LIN {X 0,Y 60.653,Z 1002.09,A -85,B 0,C 180,E1 2720.013,E2 2720.013} C_VEL
LIN {X 0,Y 76.749,Z 998.307,A -85,B 0,C 180,E1 2712.299,E2 2712.299} C_VEL
LIN {X 0,Y 92.827,Z 993.043,A -85,B 0,C 180,E1 2707.719,E2 2707.719} C_VEL
LIN {X 0,Y 109.349,Z 985.916,A -85,B 0,C 180,E1 2704.684,E2 2704.684} C_VEL
LIN {X 0,Y 120.443,Z 980.063,A -85,B 0,C 180,E1 2703.187,E2 2703.187} C_VEL
LIN {X 0,Y 109.037,Z 985.343,A -85,B 0,C 180,E1 2701.127,E2 2701.127} C_VEL
LIN {X 0,Y 102.027,Z 988.229,A -85,B 0,C 180,E1 2700.205,E2 2700.205} C_VEL
LIN {X 0,Y 85.588,Z 993.654,A -85,B 0,C 180,E1 2699.608,E2 2699.608} C_VEL
LIN {X 0,Y 77.632,Z 995.551,A -85,B 0,C 180,E1 2698.509,E2 2698.509} C_VEL
LIN {X 0,Y 75.592,Z 995.92,A -85,B 0,C 180,E1 2697.928,E2 2697.928} C_VEL
LIN {X 0,Y 59.701,Z 997.838,A -85,B 0,C 180,E1 2691.151,E2 2691.151} C_VEL
LIN {X 0,Y 45.629,Z 997.877,A -85,B 0,C 180,E1 2680.427,E2 2680.427} C_VEL
LIN {X 0,Y 33.755,Z 996.072,A -85,B 0,C 180,E1 2660.363,E2 2660.363} C_VEL
LIN {X 0,Y 28.785,Z 992.656,A -85,B 0,C 180,E1 2630.292,E2 2630.292} C_VEL
LIN {X 0,Y 32.409,Z 987.446,A -85,B 0,C 180,E1 2599.329,E2 2599.329} C_VEL
LIN {X 0,Y 42.338,Z 980.363,A -85,B 0,C 180,E1 2578.694,E2 2578.694} C_VEL
LIN {X 0,Y 54.402,Z 971.765,A -85,B 0,C 180,E1 2567.152,E2 2567.152} C_VEL
LIN {X 0,Y 66.783,Z 961.6,A -85,B 0,C 180,E1 2560.218,E2 2560.218} C_VEL
LIN {X 0,Y 78.97,Z 949.788,A -85,B 0,C 180,E1 2555.623,E2 2555.623} C_VEL
LIN {X 0,Y 89.724,Z 937.203,A -85,B 0,C 180,E1 2552.576,E2 2552.576} C_VEL
LIN {X 0,Y 99.614,Z 923.075,A -85,B 0,C 180,E1 2550.318,E2 2550.318} C_VEL
LIN {X 0,Y 108.255,Z 907.797,A -85,B 0,C 180,E1 2548.663,E2 2548.663} C_VEL
LIN {X 0,Y 114.969,Z 892.51,A -85,B 0,C 180,E1 2547.49,E2 2547.49} C_VEL
LIN {X 0,Y 120.607,Z 875.116,A -85,B 0,C 180,E1 2546.545,E2 2546.545} C_VEL
LIN {X 0,Y 124.343,Z 857.735,A -85,B 0,C 180,E1 2545.892,E2 2545.892} C_VEL
LIN {X 0,Y 132.685,Z 790.079,A -85,B 0,C 180,E1 2544.548,E2 2544.548} C_VEL
LIN {X 0,Y 132.195,Z 786.817,A -85,B 0,C 180,E1 2541.513,E2 2541.513} C_VEL
LIN {X 0,Y 131.977,Z 784.886,A -85,B 0,C 180,E1 2539.013,E2 2539.013} C_VEL
LIN {X 0,Y 131.942,Z 783.505,A -85,B 0,C 180,E1 2534.932,E2 2534.932} C_VEL
LIN {X 0,Y 132.207,Z 783.997,A -85,B 0,C 180,E1 2531.12,E2 2531.12} C_VEL
LIN {X 0,Y 132.675,Z 785.81,A -85,B 0,C 180,E1 2528.015,E2 2528.015} C_VEL
LIN {X 0,Y 133.455,Z 788.917,A -85,B 0,C 180,E1 2524.728,E2 2524.728} C_VEL
LIN {X 0,Y 133.681,Z 790.106,A -85,B 0,C 180,E1 2523.881,E2 2523.881} C_VEL
LIN {X 0,Y 124.607,Z 863.761,A -85,B 0,C 180,E1 2522.537,E2 2522.537} C_VEL
LIN {X 0,Y 120.434,Z 881.969,A -85,B 0,C 180,E1 2522.002,E2 2522.002} C_VEL
LIN {X 0,Y 115.02,Z 897.971,A -85,B 0,C 180,E1 2521.383,E2 2521.383} C_VEL
LIN {X 0,Y 107.621,Z 914.175,A -85,B 0,C 180,E1 2520.533,E2 2520.533} C_VEL
LIN {X 0,Y 98.541,Z 929.75,A -85,B 0,C 180,E1 2519.263,E2 2519.263} C_VEL
LIN {X 0,Y 88.081,Z 944.264,A -85,B 0,C 180,E1 2517.398,E2 2517.398} C_VEL
LIN {X 0,Y 76.332,Z 957.549,A -85,B 0,C 180,E1 2514.586,E2 2514.586} C_VEL
LIN {X 0,Y 63.894,Z 969.277,A -85,B 0,C 180,E1 2510.371,E2 2510.371} C_VEL
LIN {X 0,Y 51.107,Z 979.561,A -85,B 0,C 180,E1 2503.47,E2 2503.47} C_VEL
LIN {X 0,Y 38.783,Z 988.262,A -85,B 0,C 180,E1 2491.235,E2 2491.235} C_VEL
LIN {X 0,Y 29.178,Z 995.42,A -85,B 0,C 180,E1 2467.992,E2 2467.992} C_VEL
LIN {X 0,Y 27.175,Z 1000.596,A -85,B 0,C 180,E1 2434.224,E2 2434.224} C_VEL
LIN {X 0,Y 27.841,Z 1001.338,A -85,B 0,C 180,E1 2427.946,E2 2427.946} C_VEL
LIN {X 0,Y 30.091,Z 1003.083,A -85,B 0,C 180,E1 2388.356,E2 2388.356} C_VEL
LIN {X 0,Y 42.638,Z 1002.936,A -85,B 0,C 180,E1 2363.864,E2 2363.864} C_VEL
LIN {X 0,Y 59.278,Z 1000.831,A -85,B 0,C 180,E1 2351.965,E2 2351.965} C_VEL
LIN {X 0,Y 77.369,Z 996.828,A -85,B 0,C 180,E1 2345.69,E2 2345.69} C_VEL
LIN {X 0,Y 92.858,Z 991.915,A -85,B 0,C 180,E1 2342.506,E2 2342.506} C_VEL
LIN {X 0,Y 77.018,Z 995.662,A -85,B 0,C 180,E1 2338.389,E2 2338.389} C_VEL
LIN {X 0,Y 75.592,Z 995.92,A -85,B 0,C 180,E1 2337.928,E2 2337.928} C_VEL
LIN {X 0,Y 68.255,Z 997.161,A -85,B 0,C 180,E1 2336.138,E2 2336.138} C_VEL
LIN {X 0,Y 51.751,Z 999.008,A -85,B 0,C 180,E1 2333.791,E2 2333.791} C_VEL
LIN {X 0,Y 43.257,Z 999.163,A -85,B 0,C 180,E1 2330.629,E2 2330.629} C_VEL
LIN {X 0,Y 41.305,Z 999.049,A -85,B 0,C 180,E1 2329.203,E2 2329.203} C_VEL
LIN {X 0,Y 27.352,Z 997.144,A -85,B 0,C 180,E1 2309.214,E2 2309.214} C_VEL
LIN {X 0,Y 20.883,Z 993.753,A -85,B 0,C 180,E1 2272.517,E2 2272.517} C_VEL
LIN {X 0,Y 25.444,Z 988.485,A -85,B 0,C 180,E1 2231.673,E2 2231.673} C_VEL
LIN {X 0,Y 37.244,Z 981.364,A -85,B 0,C 180,E1 2209.882,E2 2209.882} C_VEL
LIN {X 0,Y 49.819,Z 973.257,A -85,B 0,C 180,E1 2199.962,E2 2199.962} C_VEL
LIN {X 0,Y 62.789,Z 963.343,A -85,B 0,C 180,E1 2194.097,E2 2194.097} C_VEL
LIN {X 0,Y 75.306,Z 951.859,A -85,B 0,C 180,E1 2190.338,E2 2190.338} C_VEL
LIN {X 0,Y 86.989,Z 938.866,A -85,B 0,C 180,E1 2187.739,E2 2187.739} C_VEL
LIN {X 0,Y 97.26,Z 924.717,A -85,B 0,C 180,E1 2185.901,E2 2185.901} C_VEL
LIN {X 0,Y 106.1,Z 909.608,A -85,B 0,C 180,E1 2184.575,E2 2184.575} C_VEL
LIN {X 0,Y 112.962,Z 894.711,A -85,B 0,C 180,E1 2183.634,E2 2183.634} C_VEL
LIN {X 0,Y 118.75,Z 877.722,A -85,B 0,C 180,E1 2182.859,E2 2182.859} C_VEL
LIN {X 0,Y 122.816,Z 860.067,A -85,B 0,C 180,E1 2182.285,E2 2182.285} C_VEL
LIN {X 0,Y 130.037,Z 803.511,A -85,B 0,C 180,E1 2181.336,E2 2181.336} C_VEL
LIN {X 0,Y 131.077,Z 794.946,A -85,B 0,C 180,E1 2181.139,E2 2181.139} C_VEL
LIN {X 0,Y 130.91,Z 792.632,A -85,B 0,C 180,E1 2178.25,E2 2178.25} C_VEL
LIN {X 0,Y 130.947,Z 791.448,A -85,B 0,C 180,E1 2174.595,E2 2174.595} C_VEL
LIN {X 0,Y 131.157,Z 791.938,A -85,B 0,C 180,E1 2171.433,E2 2171.433} C_VEL
LIN {X 0,Y 131.529,Z 793.772,A -85,B 0,C 180,E1 2168.526,E2 2168.526} C_VEL
LIN {X 0,Y 131.748,Z 795.084,A -85,B 0,C 180,E1 2167.209,E2 2167.209} C_VEL
LIN {X 0,Y 123.138,Z 863.302,A -85,B 0,C 180,E1 2166.178,E2 2166.178} C_VEL
LIN {X 0,Y 118.848,Z 881.619,A -85,B 0,C 180,E1 2165.757,E2 2165.757} C_VEL
LIN {X 0,Y 112.966,Z 898.485,A -85,B 0,C 180,E1 2165.279,E2 2165.279} C_VEL
LIN {X 0,Y 105.338,Z 914.598,A -85,B 0,C 180,E1 2164.672,E2 2164.672} C_VEL
LIN {X 0,Y 96.197,Z 929.815,A -85,B 0,C 180,E1 2163.771,E2 2163.771} C_VEL
LIN {X 0,Y 85.566,Z 944.072,A -85,B 0,C 180,E1 2162.411,E2 2162.411} C_VEL
LIN {X 0,Y 73.493,Z 957.227,A -85,B 0,C 180,E1 2160.305,E2 2160.305} C_VEL
LIN {X 0,Y 60.081,Z 969.265,A -85,B 0,C 180,E1 2156.913,E2 2156.913} C_VEL
LIN {X 0,Y 46.541,Z 979.31,A -85,B 0,C 180,E1 2151.224,E2 2151.224} C_VEL
LIN {X 0,Y 32.97,Z 987.831,A -85,B 0,C 180,E1 2140.082,E2 2140.082} C_VEL
LIN {X 0,Y 21.61,Z 994.812,A -85,B 0,C 180,E1 2113.957,E2 2113.957} C_VEL
LIN {X 0,Y 19.732,Z 999.841,A -85,B 0,C 180,E1 2066.737,E2 2066.737} C_VEL
LIN {X 0,Y 23.96,Z 1001.639,A -85,B 0,C 180,E1 2017.55,E2 2017.55} C_VEL
LIN {X 0,Y 39.12,Z 1001.702,A -85,B 0,C 180,E1 1993.786,E2 1993.786} C_VEL
LIN {X 0,Y 57.155,Z 999.903,A -85,B 0,C 180,E1 1984.344,E2 1984.344} C_VEL
LIN {X 0,Y 66.019,Z 998.339,A -85,B 0,C 180,E1 1981.724,E2 1981.724} C_VEL
LIN {X 0,Y 50.166,Z 999.311,A -85,B 0,C 180,E1 1975.222,E2 1975.222} C_VEL
LIN {X 0,Y 41.305,Z 999.049,A -85,B 0,C 180,E1 1969.203,E2 1969.203} C_VEL
LIN {X 0,Y 34.357,Z 998.611,A -85,B 0,C 180,E1 1963.944,E2 1963.944} C_VEL
LIN {X 0,Y 20.106,Z 997.162,A -85,B 0,C 180,E1 1949.983,E2 1949.983} C_VEL
LIN {X 0,Y 13.717,Z 995.406,A -85,B 0,C 180,E1 1926.437,E2 1926.437} C_VEL
LIN {X 0,Y 12.976,Z 994.699,A -85,B 0,C 180,E1 1915.311,E2 1915.311} C_VEL
LIN {X 0,Y 19.259,Z 989.522,A -85,B 0,C 180,E1 1858.718,E2 1858.718} C_VEL
LIN {X 0,Y 33.288,Z 982.367,A -85,B 0,C 180,E1 1838.646,E2 1838.646} C_VEL
LIN {X 0,Y 46.778,Z 974.342,A -85,B 0,C 180,E1 1831.237,E2 1831.237} C_VEL
LIN {X 0,Y 60.595,Z 964.276,A -85,B 0,C 180,E1 1826.991,E2 1826.991} C_VEL
LIN {X 0,Y 73.542,Z 952.771,A -85,B 0,C 180,E1 1824.363,E2 1824.363} C_VEL
LIN {X 0,Y 85.525,Z 939.759,A -85,B 0,C 180,E1 1822.541,E2 1822.541} C_VEL
LIN {X 0,Y 96.011,Z 925.604,A -85,B 0,C 180,E1 1821.238,E2 1821.238} C_VEL
LIN {X 0,Y 105.005,Z 910.497,A -85,B 0,C 180,E1 1820.292,E2 1820.292} C_VEL
LIN {X 0,Y 111.98,Z 895.625,A -85,B 0,C 180,E1 1819.606,E2 1819.606} C_VEL
LIN {X 0,Y 117.862,Z 878.714,A -85,B 0,C 180,E1 1819.024,E2 1819.024} C_VEL
LIN {X 0,Y 122.059,Z 860.873,A -85,B 0,C 180,E1 1818.568,E2 1818.568} C_VEL
LIN {X 0,Y 129.056,Z 807.041,A -85,B 0,C 180,E1 1817.844,E2 1817.844} C_VEL
LIN {X 0,Y 129.873,Z 800.465,A -85,B 0,C 180,E1 1817.7,E2 1817.7} C_VEL
LIN {X 0,Y 129.958,Z 799.398,A -85,B 0,C 180,E1 1814.203,E2 1814.203} C_VEL
LIN {X 0,Y 130.128,Z 799.983,A -85,B 0,C 180,E1 1811.525,E2 1811.525} C_VEL
LIN {X 0,Y 130.184,Z 800.71,A -85,B 0,C 180,E1 1810.617,E2 1810.617} C_VEL
LIN {X 0,Y 122.208,Z 862.683,A -85,B 0,C 180,E1 1809.894,E2 1809.894} C_VEL
LIN {X 0,Y 117.878,Z 880.934,A -85,B 0,C 180,E1 1809.604,E2 1809.604} C_VEL
LIN {X 0,Y 111.964,Z 897.733,A -85,B 0,C 180,E1 1809.318,E2 1809.318} C_VEL
LIN {X 0,Y 104.272,Z 913.833,A -85,B 0,C 180,E1 1809.001,E2 1809.001} C_VEL
LIN {X 0,Y 94.795,Z 929.39,A -85,B 0,C 180,E1 1808.493,E2 1808.493} C_VEL
LIN {X 0,Y 84.256,Z 943.252,A -85,B 0,C 180,E1 1807.728,E2 1807.728} C_VEL
LIN {X 0,Y 72.464,Z 955.886,A -85,B 0,C 180,E1 1806.539,E2 1806.539} C_VEL
LIN {X 0,Y 59.185,Z 967.561,A -85,B 0,C 180,E1 1804.61,E2 1804.61} C_VEL
LIN {X 0,Y 45.005,Z 977.757,A -85,B 0,C 180,E1 1801.137,E2 1801.137} C_VEL
LIN {X 0,Y 30.174,Z 986.37,A -85,B 0,C 180,E1 1793.813,E2 1793.813} C_VEL
LIN {X 0,Y 15.929,Z 993.428,A -85,B 0,C 180,E1 1771.509,E2 1771.509} C_VEL
LIN {X 0,Y 11.636,Z 998.326,A -85,B 0,C 180,E1 1703.529,E2 1703.529} C_VEL
LIN {X 0,Y 20.92,Z 1000.281,A -85,B 0,C 180,E1 1637.096,E2 1637.096} C_VEL
LIN {X 0,Y 39.002,Z 1000.384,A -85,B 0,C 180,E1 1621.252,E2 1621.252} C_VEL
LIN {X 0,Y 39.996,Z 1000.332,A -85,B 0,C 180,E1 1620.714,E2 1620.714} C_VEL
LIN {X 0,Y 23.703,Z 998.518,A -85,B 0,C 180,E1 1605.957,E2 1605.957} C_VEL
LIN {X 0,Y 13.256,Z 995.1,A -85,B 0,C 180,E1 1561.861,E2 1561.861} C_VEL
LIN {X 0,Y 12.976,Z 994.699,A -85,B 0,C 180,E1 1555.311,E2 1555.311} C_VEL
LIN {X 0,Y 13.117,Z 992.68,A -85,B 0,C 180,E1 1522.061,E2 1522.061} C_VEL
LIN {X 0,Y 20.049,Z 988.479,A -85,B 0,C 180,E1 1478.299,E2 1478.299} C_VEL
LIN {X 0,Y 27.105,Z 985.199,A -85,B 0,C 180,E1 1467.299,E2 1467.299} C_VEL
LIN {X 0,Y 30.994,Z 983.298,A -85,B 0,C 180,E1 1465.033,E2 1465.033} C_VEL
LIN {X 0,Y 46.16,Z 974.608,A -85,B 0,C 180,E1 1461.337,E2 1461.337} C_VEL
LIN {X 0,Y 60.41,Z 964.371,A -85,B 0,C 180,E1 1459.359,E2 1459.359} C_VEL
LIN {X 0,Y 73.627,Z 952.692,A -85,B 0,C 180,E1 1458.078,E2 1458.078} C_VEL
LIN {X 0,Y 85.291,Z 940.003,A -85,B 0,C 180,E1 1457.168,E2 1457.168} C_VEL
LIN {X 0,Y 95.916,Z 925.717,A -85,B 0,C 180,E1 1456.451,E2 1456.451} C_VEL
LIN {X 0,Y 105.013,Z 910.452,A -85,B 0,C 180,E1 1455.914,E2 1455.914} C_VEL
LIN {X 0,Y 112.462,Z 894.241,A -85,B 0,C 180,E1 1455.47,E2 1455.47} C_VEL
LIN {X 0,Y 118.411,Z 876.546,A -85,B 0,C 180,E1 1455.086,E2 1455.086} C_VEL
LIN {X 0,Y 122.26,Z 859.199,A -85,B 0,C 180,E1 1454.782,E2 1454.782} C_VEL
LIN {X 0,Y 128.956,Z 807.335,A -85,B 0,C 180,E1 1454.255,E2 1454.255} C_VEL
LIN {X 0,Y 128.923,Z 807.647,A -85,B 0,C 180,E1 1454.084,E2 1454.084} C_VEL
LIN {X 0,Y 121.758,Z 862.27,A -85,B 0,C 180,E1 1453.65,E2 1453.65} C_VEL
LIN {X 0,Y 117.384,Z 880.469,A -85,B 0,C 180,E1 1453.495,E2 1453.495} C_VEL
LIN {X 0,Y 111.528,Z 896.981,A -85,B 0,C 180,E1 1453.411,E2 1453.411} C_VEL
LIN {X 0,Y 103.607,Z 913.441,A -85,B 0,C 180,E1 1453.393,E2 1453.393} C_VEL
LIN {X 0,Y 94.273,Z 928.636,A -85,B 0,C 180,E1 1453.324,E2 1453.324} C_VEL
LIN {X 0,Y 83.452,Z 942.704,A -85,B 0,C 180,E1 1453.16,E2 1453.16} C_VEL
LIN {X 0,Y 70.758,Z 956.024,A -85,B 0,C 180,E1 1452.827,E2 1452.827} C_VEL
LIN {X 0,Y 57.309,Z 967.505,A -85,B 0,C 180,E1 1452.297,E2 1452.297} C_VEL
LIN {X 0,Y 42.814,Z 977.451,A -85,B 0,C 180,E1 1451.215,E2 1451.215} C_VEL
LIN {X 0,Y 26.668,Z 986.22,A -85,B 0,C 180,E1 1448.63,E2 1448.63} C_VEL
LIN {X 0,Y 11.002,Z 992.806,A -85,B 0,C 180,E1 1439.09,E2 1439.09} C_VEL
LIN {X 0,Y 3.754,Z 996.779,A -85,B 0,C 180,E1 1324.356,E2 1324.356} C_VEL
LIN {X 0,Y 14.343,Z 998.4,A -85,B 0,C 180,E1 1258.451,E2 1258.451} C_VEL
LIN {X 0,Y 6.121,Z 994.111,A -85,B 0,C 180,E1 1150.914,E2 1150.914} C_VEL
LIN {X 0,Y 20.808,Z 988.067,A -85,B 0,C 180,E1 1110.114,E2 1110.114} C_VEL
LIN {X 0,Y 30.994,Z 983.298,A -85,B 0,C 180,E1 1105.033,E2 1105.033} C_VEL
LIN {X 0,Y 33.822,Z 985.097,A -85,B 0,C 180,E1 1104.141,E2 1104.141} C_VEL
LIN {X 0,Y 33.822,Z 1084,A -85,B 0,C 180,E1 1104.141,E2 1104.141} C_VEL
LIN {X 0,Y 33.822,Z 1084,A -85,B 0,C 180,E1 1104.141,E2 1104.141}

QRS_NEXT_CUT()

QRS_NEXT()
QRS_HOME()

END
